FUNCTION_BLOCK FB_BaseTopElementDecoratorParent EXTENDS FB_BaseGroupElementDecoratorParent IMPLEMENTS ITF_BaseTopElementDecoratorParent
VAR
	itfTopElement				: ITF_BaseTopElement;
END_VAR

(*			
	EVERDE sp. z o.o.
	Rafał Osajda		24.03.2025		TC 4024.66
	Definicja nowego zgłoszenia
*)
METHOD PUBLIC EventsDefinition : BOOL
EventsDefinition		:= THIS^.itfTopElement.EventsDefinition ();
END_METHOD

(*			
	EVERDE sp. z o.o.
	Rafał Osajda		27.03.2025		TC 4024.66
	Obsluga bledow sprawdzanie czy jakis blad sie nei pojawil i ustawienie stanu lub wylaczenie
*)
METHOD PUBLIC ExecuteEveryCycle_Error
VAR_INPUT
END_VAR
THIS^.itfTopElement.ExecuteEveryCycle_Error ();
END_METHOD

(*			
	EVERDE sp. z o.o.
	Rafał Osajda		27.03.2025		TC 4024.66
	Wywolanie co cykl operacji 
*)
METHOD PUBLIC ExecuteEveryCycle_Operation
VAR_INPUT
END_VAR
THIS^.itfTopElement.ExecuteEveryCycle_Operation ();
END_METHOD

(*			
	EVERDE sp. z o.o.
	Rafał Osajda		27.03.2025		TC 4024.66
	Aktualizacja flag 
*)
METHOD PUBLIC ExecuteEveryCycle_Status
VAR_INST
END_VAR
THIS^.itfTopElement.ExecuteEveryCycle_Status ();
END_METHOD

(*			
	EVERDE sp. z o.o.
	Rafał Osajda		27.03.2025		TC 4024.66
	Testowanie czy nei pojawil sie jakis rozkaz i uruchomienie odpowiednich operacji
*)
METHOD PUBLIC ExecuteEveryCycle_Test
VAR_INPUT
END_VAR
THIS^.itfTopElement.ExecuteEveryCycle_Test ();
END_METHOD

METHOD FB_init : BOOL
VAR_INPUT
	bInitRetains : BOOL; // if TRUE, the retain variables are initialized (warm start / cold start)
	bInCopyCode : BOOL;  // if TRUE, the instance afterwards gets moved into the copy code (online change)
	fbToDecorate		: ITF_DecoratedElement;
END_VAR
THIS^.itfTopElement	:= fbToDecorate.GetITFTopElement ();
END_METHOD

(*			
	EVERDE sp. z o.o.
	Rafał Osajda		03.10.2025		TC 4024.66
	
*)
METHOD PUBLIC FirstCycle : BOOL
VAR_INPUT
END_VAR
FirstCycle				:= THIS^.itfTopElement.FirstCycle ();
END_METHOD

METHOD PUBLIC GetCode : STRING
VAR_INPUT
END_VAR
GetCode			:= THIS^.itfTopElement.GetCode ();
END_METHOD

(*			
	EVERDE sp. z o.o.
	Rafał Osajda		30.04.2025		TC 4024.66
	Zwraca czy element jest czymś zajety
*)
METHOD PUBLIC GetDoNothing : BOOL
GetDoNothing		:= THIS^.itfTopElement.GetDoNothing ();
END_METHOD

METHOD PUBLIC GetID : UINT
VAR_INPUT
END_VAR
GetID		:= THIS^.itfTopElement.GetID ();
END_METHOD

METHOD PUBLIC GetIdentyfier : ST_BaseElementIdentifier
VAR_INPUT
END_VAR
GetIdentyfier		:= THIS^.itfTopElement.GetIdentyfier ();
END_METHOD

METHOD PUBLIC GetName : ST_BaseLabel
VAR_INPUT
END_VAR
GetName		:= THIS^.itfTopElement.GetName ();
END_METHOD

(*			
	EVERDE sp. z o.o.
	Rafał Osajda		30.04.2025		TC 4024.66
	Zwraca czy element jest w pozycji 0 - referencyjnej
*)
METHOD PUBLIC GetPosition0 : BOOL
GetPosition0	:= THIS^.itfTopElement.GetPosition0 ();
END_METHOD

METHOD PUBLIC GetType : E_BaseElementType
VAR_INPUT
END_VAR
GetType		:= THIS^.itfTopElement.GetType ();
END_METHOD

(*			
	EVERDE sp. z o.o.
	Rafał Osajda		31.03.2025		TC 4024.66
	Flaga że w tej sesji pracy maszyny element został już wybazowany
*)
METHOD PUBLIC HomingGetDone : BOOL
VAR_INPUT
END_VAR
HomingGetDone	:= THIS^.itfTopElement.HomingGetDone ();
END_METHOD

(*			
	EVERDE sp. z o.o.
	Rafał Osajda		11.04.2025		TC 4024.66
	Zwraca czy bazowanie jest potrzebne
*)
METHOD PUBLIC HomingGetIsNeeded : BOOL
VAR_INPUT
END_VAR
HomingGetIsNeeded	:= THIS^.itfTopElement.HomingGetIsNeeded ();
END_METHOD

(*			
	EVERDE sp. z o.o.
	Rafał Osajda		27.05.2025		TC 4024.66
	Uruchomienie metody bazowania
*)
METHOD PUBLIC HomingStart
VAR_INPUT
END_VAR
THIS^.itfTopElement.HomingStart ();
END_METHOD

METHOD PUBLIC IsValidCommonData : BOOL
VAR_INPUT
END_VAR
IsValidCommonData			:= THIS^.itfTopElement.IsValidCommonData ();
END_METHOD

(*			
	EVERDE sp. z o.o.
	Rafał Osajda		07.10.2025		TC 4024.66
	Dodpisywanie się do listy logera
*)
METHOD PUBLIC JoinTheLogger : BOOL
VAR_INPUT
END_VAR
JoinTheLogger	:= THIS^.itfTopElement.JoinTheLogger ();
END_METHOD

METHOD PUBLIC LinkCommonData : BOOL
VAR_INPUT
	stCommonData				: REFERENCE TO ST_BaseCommonData;
END_VAR
LinkCommonData			:= THIS^.itfTopElement.LinkCommonData (stCommonData := stCommonData);
END_METHOD

METHOD PUBLIC LinkSS1 : BOOL
VAR_INPUT
	fbSS1			: ITF_BaseFlagGet;
END_VAR
LinkSS1		:= THIS^.itfTopElement.LinkSS1 (fbSS1 := fbSS1);
END_METHOD

METHOD PUBLIC LinkSTO : BOOL
VAR_INPUT
	fbSTO			: ITF_BaseFlagGet;
END_VAR
LinkSTO		:= THIS^.itfTopElement.LinkSTO (fbSTO := fbSTO);
END_METHOD

(*			
	EVERDE sp. z o.o.
	Rafał Osajda		31.03.2025		TC 4024.66
	Zwraca status zasilania	
*)
METHOD PUBLIC PowerGetStatus : BOOL
VAR_INPUT
END_VAR
PowerGetStatus		:= THIS^.itfTopElement.PowerGetStatus ();
END_METHOD

(*			
	EVERDE sp. z o.o.
	Rafał Osajda		31.03.2025		TC 4024.66
	Wyłączenie zasilania
*)
METHOD PUBLIC PowerTurnOff : BOOL
VAR_INPUT
END_VAR
PowerTurnOff		:= THIS^.itfTopElement.PowerTurnOff ();
END_METHOD

(*			
	EVERDE sp. z o.o.
	Rafał Osajda		31.03.2025		TC 4024.66
	Uruchomienie zasialania
*)
METHOD PUBLIC PowerTurnOn
VAR_INPUT
END_VAR
THIS^.itfTopElement.PowerTurnOn ();
END_METHOD

METHOD PUBLIC Reset : BOOL
VAR_INPUT
END_VAR
Reset	:= THIS^.itfTopElement.Reset ();
END_METHOD

METHOD PUBLIC ResetGetBusy : BOOL
VAR_INPUT
END_VAR
ResetGetBusy		:= THIS^.itfTopElement.ResetGetBusy ();
END_METHOD

METHOD PUBLIC ResetGetStatus : BOOL
VAR_INPUT
END_VAR
ResetGetStatus			:= THIS^.itfTopElement.ResetGetStatus ();
END_METHOD

METHOD PUBLIC SetCode
VAR_INPUT
	sCode							: STRING;
	sAdd							: STRING;
END_VAR
THIS^.itfTopElement.SetCode (sCode := sCode, sAdd := sAdd);
END_METHOD

(*			
	EVERDE sp. z o.o.
	Rafał Osajda		03.10.2025		TC 4024.66
	nadawanie unikalnych ID dla zdarzeń
*)
METHOD PUBLIC SetEventsIDs : UINT
VAR_INPUT
	uiNewID		: UINT;
END_VAR
SetEventsIDs		:= THIS^.itfTopElement.SetEventsIDs (uiNewID := uiNewID);
END_METHOD

METHOD PUBLIC SetID : UINT
VAR_INPUT
	uiID					: UINT;
END_VAR
SetID		:= THIS^.itfTopElement.SetID (uiID := uiID);
END_METHOD

METHOD PUBLIC SetName
VAR_INPUT
	stName				: ST_BaseLabel;
END_VAR
THIS^.itfTopElement.SetName (stName := stName);
END_METHOD

METHOD PUBLIC SetType
VAR_INPUT
	eType					: E_BaseElementType;
END_VAR
THIS^.itfTopElement.SetType (eType := eType);
END_METHOD

END_FUNCTION_BLOCK

(* stored: Version 1.1.0.1
   POU FB_BaseTopElementDecoratorParent: Id {e103fea3-a4b4-0fb2-23f5-e57c59155c7a}, SpecialFunc None
   Folder Bazowanie: Id {263db5f0-3a56-09ff-0a9d-c1e15abec839}
   Folder Events: Id {7e2b3539-94ac-0848-1dec-524615c47062}
   Folder ID: Id {cbbc977a-d53a-0d8d-1d46-a2dc57926fef}
   Folder ITF_BaseComponent: Id {23a03bd9-1942-041e-05da-dd5b6b05c7bd}
   Folder WiazanieZmiennych: Id {ec9a7be5-a160-0408-2aaf-fec9e4c8031e}
   Folder Zasilanie: Id {976f8ba9-242b-0706-3db6-722b359ecd59}
   Method EventsDefinition: Id {3c3f7f57-b1c7-05a8-1ed8-52a48a3d4fe2}
   Method ExecuteEveryCycle_Error: Id {b6969075-a994-0c38-0653-8b7cf77af3b5}
   Method ExecuteEveryCycle_Operation: Id {c3ce2a7b-b612-0d1d-1efa-fdc1186cdbf6}
   Method ExecuteEveryCycle_Status: Id {9374fa9e-5e3a-0d70-28e4-07c3f08616a7}
   Method ExecuteEveryCycle_Test: Id {9fd84e0f-da37-05de-3361-260ccbe56b66}
   Method FB_init: Id {b8cb3433-cf7a-0e4d-10cb-6b629cb40e90}
   Method FirstCycle: Id {2a7242df-8b1b-047e-3cff-aab1b65306bd}
   Method GetCode: Id {c54f8afb-50c0-0057-1911-304a7c944824}
   Method GetDoNothing: Id {f0841806-0d5c-0217-072e-1bcf0bbfbdf0}
   Method GetID: Id {c7f9633d-0f1a-0d52-1e62-45c3cab72e30}
   Method GetIdentyfier: Id {fafe425e-aa69-0814-231e-ef880b6d7b85}
   Method GetName: Id {a098d7ee-78be-05ca-02e8-3ddc38ba1179}
   Method GetPosition0: Id {c94a2fcb-40aa-0c72-0ae4-b72f06c666de}
   Method GetType: Id {ed04e64e-7559-090d-2159-1c7eefea1008}
   Method HomingGetDone: Id {ca90527b-f800-0fbb-37dc-8b70efe79b36}
   Method HomingGetIsNeeded: Id {bd51ebf7-c238-0521-3353-b5493fb9b1bc}
   Method HomingStart: Id {38dbdcec-1ff3-0725-3b4d-ee8050aa2e02}
   Method IsValidCommonData: Id {de1af751-abe1-06bd-289b-a3350d1444de}
   Method JoinTheLogger: Id {6f630d1a-2ac1-042e-015f-130054ad0c0d}
   Method LinkCommonData: Id {9f5ce9b5-044d-03ff-34a4-ac5bdd68d213}
   Method LinkSS1: Id {9611b700-b131-08c5-1963-13ee75fb3ede}
   Method LinkSTO: Id {e5d184c8-1371-0bbc-18fd-2e02c87486b8}
   Method PowerGetStatus: Id {193116b8-1ea4-0185-2ca8-8288226c4556}
   Method PowerTurnOff: Id {7bfe67cc-0910-0a5a-3b7f-9b8cf2cc0d8a}
   Method PowerTurnOn: Id {14b58fa7-ceea-0d05-3978-51e82a563423}
   Method Reset: Id {6e38683c-ba43-0a1e-0662-6e7a62e04084}
   Method ResetGetBusy: Id {aa7b660b-aede-0070-1e44-0f28aa3bc68f}
   Method ResetGetStatus: Id {9cb205dc-5834-0506-036a-4cde0a57e89a}
   Method SetCode: Id {e204e6d8-7820-0332-32ad-2a74665cec3a}
   Method SetEventsIDs: Id {1805e4e5-d1a2-06de-2c4b-1302b367e8eb}
   Method SetID: Id {37ca3965-00d2-02a5-0599-806cebaa187b}
   Method SetName: Id {1207a2fa-8a60-0d95-26a9-6f08411ca7fe}
   Method SetType: Id {9c976999-ec4a-09df-23df-d4faafb92caf} *)
